Universal Robots PolyScope program: Move.urp

Program Move (installation=default directory=/programs/archive createdIn=3.3.0.145 lastSavedIn=5.11.5.1010327 robotSerialNumber=20215500677)
Calibrated DH parameters: a=[0.000204, -0.239222, -0.391845, -0.000001, 0.000022, 0]; d=[0.162722, -355.808559, 353.37206, 2.570385, 0.099741, 0.099629]; alpha=[1.571124, 0.000988, 0.008295, 1.568963, -1.570303, 0]; deltaTheta=[0, -0.973091, 7.204745, 0.05153, 0, 0]
Robot Program (runOnlyOnce=true)
  Script file /programs/Move.script
    | def Move() :
    | 
    | set_payload(1.29)
    | set_tcp(p[0,0,0,0,0,0])
    | movep(p[0.211331,0,0.98005,2.221441,2.221441,0], a=10, v=0.25, r=0.001)
    | 
    | end
    | 
    | 
    | Move()
